Omron CX-Programmer project 新工程 (CX-Programmer 9.73)

# PLC 新PLC1: CPM2* 

## Global symbols (name address type ; comment)
0.00 BOOL  ; 横限1
0.01 BOOL  ; 横限2
0.02 BOOL  ; 横限3
0.03 BOOL  ; 横限4
0.04 BOOL  ; 横限5
0.05 BOOL  ; 二层上限1
0.06 BOOL  ; 二层上限2
0.07 BOOL  ; 二层上限3
0.08 BOOL  ; 二层上限4
0.09 BOOL  ; 二层下限1
0.10 BOOL  ; 二层下限2
0.11 BOOL  ; 二层下限3
10.00 BOOL  ; 总接触器1
10.01 BOOL  ; 总接触器2
10.02 BOOL  ; 1号可升降
10.03 BOOL  ; 2号可升降
10.04 BOOL  ; 3号可升降
10.06 BOOL  ; 4号可升降
11.00 BOOL  ; 5号横移
11.01 BOOL  ; 6号横移
11.02 BOOL  ; 7号横移
11.03 BOOL  ; 8号横移
11.04 BOOL  ; 9号可升降
11.06 BOOL  ; 10号可升降
12.00 BOOL  ; 11号可升降
12.01 BOOL  ; 12号可升降
12.02 BOOL  ; 故障报警
12.03 BOOL  ; 运行警示
12.04 BOOL  ; 左围栏升降
12.05 BOOL  ; 右围栏升降
12.06 BOOL  ; 围栏总上升
12.07 BOOL  ; 围栏总下降
16.00 BOOL  ; 手1
16.01 BOOL  ; 手2
16.02 BOOL  ; 手3
16.03 BOOL  ; 手4
16.04 BOOL  ; 手5
16.05 BOOL  ; 手6
16.06 BOOL  ; 手7
16.07 BOOL  ; 手8
16.08 BOOL  ; 手9
17.00 BOOL  ; 手动有车位输入
17.07 BOOL  ; =0
17.08 BOOL  ; >0
17.10 BOOL  ; OK
17.11 BOOL  ; ER
17.15 BOOL  ; >14
18.08 BOOL  ; 自动↑
18.09 BOOL  ; 手动↑
18.10 BOOL  ; 刷卡↑
18.13 BOOL  ; 启动延迟
18.14 BOOL  ; 自动脉冲
1.00 BOOL  ; 二层下限4
1.01 BOOL  ; 底层上限1
1.02 BOOL  ; 底层上限2
1.03 BOOL  ; 底层上限3
1.04 BOOL  ; 底层上限4
1.05 BOOL  ; 底层下限1
1.06 BOOL  ; 底层下限2
1.07 BOOL  ; 底层下限3
1.08 BOOL  ; 底层下限4
1.09 BOOL  ; 左围栏上限
1.10 BOOL  ; 右围栏上限
1.11 BOOL  ; 左围栏下限
202.01 BOOL  ; 1号卡
202.02 BOOL  ; 2号卡
202.03 BOOL  ; 3号卡
202.04 BOOL  ; 4号卡
202.05 BOOL  ; 5号卡
202.06 BOOL  ; 6号卡
202.07 BOOL  ; 7号卡
202.08 BOOL  ; 8号卡
202.09 BOOL  ; 9号卡
202.10 BOOL  ; 10号卡
202.11 BOOL  ; 11号卡
202.12 BOOL  ; 12号卡
203.02 BOOL  ; 二层可上
203.03 BOOL  ; 底层可下
203.05 BOOL  ; 二层全在上
203.06 BOOL  ; 底层全在下
203.07 BOOL  ; 升降至原位
204.00 BOOL  ; 0
204.01 BOOL  ; 1
204.02 BOOL  ; 2
204.03 BOOL  ; 3
204.04 BOOL  ; 4
204.05 BOOL  ; 5
204.06 BOOL  ; 6
204.07 BOOL  ; 7
204.08 BOOL  ; 8
204.09 BOOL  ; 9
205.04 BOOL  ; 升降
206.10 BOOL  ; 运行
206.11 BOOL  ; 故障
206.12 BOOL  ; 故障排除后启动
206.13 BOOL  ; 有故障
206.14 BOOL  ; 故障排除
206.15 BOOL  ; 故障↓
207.00 BOOL  ; 操作可
207.02 BOOL  ; 卡号
207.15 BOOL  ; 升降
208.00 BOOL  ; 自动车位号为1234
208.01 BOOL  ; 自动
208.02 BOOL  ; 在中间
208.05 BOOL  ; 自动车位号不等于1234
208.06 BOOL  ; 自动车位号不等于1234
208.07 BOOL  ; > 12
208.09 BOOL  ; ＞12，14
209.00 BOOL  ; 自动
209.01 BOOL  ; 手动
209.02 BOOL  ; 刷卡↑
209.05 BOOL  ; 刷卡
209.14 BOOL  ; 自动↑
209.15 BOOL  ; 自动车位号不等于1234↑
210.05 BOOL  ; 有四位数输入
211.00 BOOL  ; O-0
211.01 BOOL  ; 0-1
211.02 BOOL  ; 0-2
211.03 BOOL  ; 0-3
211.04 BOOL  ; 0-4
211.05 BOOL  ; 0-5
211.06 BOOL  ; 0-6
211.07 BOOL  ; 0-7
211.08 BOOL  ; 0-8
211.09 BOOL  ; 0-9
212.00 BOOL  ; 1-0
212.01 BOOL  ; 1-1
212.02 BOOL  ; 1-2
212.03 BOOL  ; 1-3
212.04 BOOL  ; 1-4
212.05 BOOL  ; 1-5
212.06 BOOL  ; 1-6
212.07 BOOL  ; 1-7
212.08 BOOL  ; 1-8
212.09 BOOL  ; 1-9
212.10 BOOL  ; F保持
212.11 BOOL  ; 左围栏S
212.12 BOOL  ; 右围栏S
213.00 BOOL  ; 2-0
213.01 BOOL  ; 2-1
213.02 BOOL  ; 2-2
213.03 BOOL  ; 2-3
213.04 BOOL  ; 2-4
213.05 BOOL  ; 2-5
213.06 BOOL  ; 2-6
213.07 BOOL  ; 2-7
213.08 BOOL  ; 2-8
213.09 BOOL  ; 2-9
213.11 BOOL  ; 左围栏X
213.12 BOOL  ; 右围栏X
214.00 BOOL  ; 3-0
214.01 BOOL  ; 3-1
214.02 BOOL  ; 3-2
214.03 BOOL  ; 3-3
214.04 BOOL  ; 3-4
214.05 BOOL  ; 3-5
214.06 BOOL  ; 3-6
214.07 BOOL  ; 3-7
214.08 BOOL  ; 3-8
214.09 BOOL  ; 3-9
216.01 BOOL  ; 1号卡2
216.02 BOOL  ; 2号卡2
216.03 BOOL  ; 3号卡2
216.04 BOOL  ; 4号卡2
216.05 BOOL  ; 5号卡2
216.06 BOOL  ; 6号卡2
216.07 BOOL  ; 7号卡2
216.08 BOOL  ; 8号卡2
216.09 BOOL  ; 9号卡2
216.10 BOOL  ; 10号卡2
216.11 BOOL  ; 11号卡2
216.12 BOOL  ; 12号卡2
217.00 BOOL  ; 升降至原位↑
217.01 BOOL  ; 到位
219.01 BOOL  ; 1号卡3
219.02 BOOL  ; 2号卡3
219.03 BOOL  ; 3号卡3
219.04 BOOL  ; 4号卡3
219.05 BOOL  ; 5号卡3
219.06 BOOL  ; 6号卡3
219.07 BOOL  ; 7号卡3
219.08 BOOL  ; 8号卡3
219.09 BOOL  ; 9号卡3
219.10 BOOL  ; 10号卡3
219.11 BOOL  ; 11号卡3
219.12 BOOL  ; 12号卡3
220.10 BOOL  ; 一位输入
220.11 BOOL  ; 二位输入
220.12 BOOL  ; 三位输入
220.13 BOOL  ; 四位输入
222.00 BOOL  ; 手10
222.01 BOOL  ; 手11
222.02 BOOL  ; 手12
222.03 BOOL  ; 手13
222.04 BOOL  ; 手14
224.00 BOOL  ; 手取1
224.01 BOOL  ; 手取2
224.02 BOOL  ; 手取3
224.03 BOOL  ; 手取4
224.04 BOOL  ; 手取5
224.05 BOOL  ; 手取6
224.06 BOOL  ; 手取7
224.07 BOOL  ; 手取8
224.08 BOOL  ; 手取9
224.09 BOOL  ; 手取10
224.10 BOOL  ; 手取11
224.12 BOOL  ; 手取12
224.13 BOOL  ; 手取13
224.14 BOOL  ; 手取14
22.00 BOOL  ; 横移过快
22.01 BOOL  ; 有故障
22.02 BOOL  ; 横移过快
22.06 BOOL  ; 横移
22.07 BOOL  ; 5号横移↓
22.08 BOOL  ; 6号横移↓
22.09 BOOL  ; 7号横移↓
22.10 BOOL  ; 8号横移↓
22.11 BOOL  ; 人车进出上升沿
22.12 BOOL  ; 延时上升沿
230.06 BOOL  ; 7Z
230.07 BOOL  ; 5Z
230.08 BOOL  ; 6Z
230.09 BOOL  ; 7Z
230.10 BOOL  ; 8Z
230.12 BOOL  ; 12Z
232.00 BOOL  ; 1S
232.01 BOOL  ; 2S
232.02 BOOL  ; 3S
232.03 BOOL  ; 4S
232.14 BOOL  ; 9S
232.15 BOOL  ; 10S
233.00 BOOL  ; 11S
233.01 BOOL  ; 12S
236.00 BOOL  ; ZD1
236.01 BOOL  ; ZD2
236.02 BOOL  ; ZD3
236.03 BOOL  ; ZD4
236.05 BOOL  ; ZD6
236.06 BOOL  ; ZD7
236.07 BOOL  ; ZD9
236.08 BOOL  ; ZD10
236.09 BOOL  ; ZD11
236.10 BOOL  ; ZD12
23.00 BOOL  ; 横移
23.01 BOOL  ; 横移
240.07 BOOL  ; 5Y
240.08 BOOL  ; 6Y
240.09 BOOL  ; 7Y
240.10 BOOL  ; 8Y
242.00 BOOL  ; 1X
242.01 BOOL  ; 2X
242.02 BOOL  ; 3X
242.03 BOOL  ; 4X
242.14 BOOL  ; 9X
242.15 BOOL  ; 10X
243.00 BOOL  ; 11X
243.01 BOOL  ; 12X
28.08 BOOL  ; > 14
2.00 BOOL  ; 右围栏下限
2.01 BOOL  ; 底层防坠落
2.02 BOOL  ; 二层松链
2.03 BOOL  ; 底层超上限
2.04 BOOL  ; 二层超上限
2.05 BOOL  ; 车高光电
2.06 BOOL  ; 人车进出
2.07 BOOL  ; 车长光电
2.08 BOOL  ; 急停
2.09 BOOL  ; 热保护
2.10 BOOL  ; 相序保护
30.00 BOOL  ; 1号在下
30.01 BOOL  ; 2号在下
30.02 BOOL  ; 3号在下
30.03 BOOL  ; 4号在下
31.01 BOOL  ; 二层总上升
31.02 BOOL  ; 二层总下降
31.03 BOOL  ; 底层总上升
31.04 BOOL  ; 底层总下降
31.05 BOOL  ; 一层总左移
31.06 BOOL  ; 一层总右移
31.07 BOOL  ; 左围栏上升
31.08 BOOL  ; 左围栏下降
31.09 BOOL  ; 右围栏上升
31.10 BOOL  ; 右围栏下降
32.02 BOOL  ; （到位）
34.00 BOOL  ; Z1
34.01 BOOL  ; Z2
34.02 BOOL  ; Z3
34.03 BOOL  ; Z4
34.04 BOOL  ; Z5
34.05 BOOL  ; Z6
34.06 BOOL  ; Z7
34.07 BOOL  ; Z8
34.08 BOOL  ; Z9
34.09 BOOL  ; Z10
34.10 BOOL  ; Z11
34.12 BOOL  ; Z12
35.15 BOOL  ; > 12
37.12 BOOL  ; 重取
40.00 BOOL  ; 0
40.01 BOOL  ; 1
40.02 BOOL  ; 2/上
40.03 BOOL  ; 3
40.04 BOOL  ; 4左
40.05 BOOL  ; 5
40.06 BOOL  ; 6右
40.07 BOOL  ; 7
40.08 BOOL  ; 8/下
40.09 BOOL  ; 9
40.10 BOOL  ; 启动
40.11 BOOL  ; 复位
40.12 BOOL  ; 手动
40.13 BOOL  ; 在中间
40.14 BOOL  ; 自动
40.15 BOOL  ; F
41.00 BOOL  ; 1号可上下
41.01 BOOL  ; 2号可上下
41.02 BOOL  ; 3号可上下
41.03 BOOL  ; 4号可上下
41.08 BOOL  ; 9号可上下
41.09 BOOL  ; 10号可上下
41.10 BOOL  ; 11号可上下
41.11 BOOL  ; 12号可上下
42.01 BOOL  ; 1号卡
42.02 BOOL  ; 2号卡
42.03 BOOL  ; 3号卡
42.04 BOOL  ; 4号卡
42.05 BOOL  ; 5号卡
42.06 BOOL  ; 6号卡
42.07 BOOL  ; 7号卡
42.08 BOOL  ; 8号卡
43.00 BOOL  ; 9号卡
43.01 BOOL  ; 10号卡
43.02 BOOL  ; 11号卡
43.03 BOOL  ; 12号卡
44.01 BOOL  ; 1号卡2
44.02 BOOL  ; 2号卡2
44.03 BOOL  ; 3号卡2
44.04 BOOL  ; 4号卡2
44.05 BOOL  ; 5号卡2
44.06 BOOL  ; 6号卡2
44.07 BOOL  ; 7号卡2
44.08 BOOL  ; 8号卡2
45.00 BOOL  ; 9号卡2
45.01 BOOL  ; 10号卡2
45.02 BOOL  ; 11号卡2
45.03 BOOL  ; 12号卡2
46.01 BOOL  ; 1号卡3
46.02 BOOL  ; 2号卡3
46.03 BOOL  ; 3号卡3
46.04 BOOL  ; 4号卡3
46.05 BOOL  ; 5号卡3
46.06 BOOL  ; 6号卡3
46.07 BOOL  ; 7号卡3
46.08 BOOL  ; 8号卡3
47.00 BOOL  ; 9号卡3
47.01 BOOL  ; 10号卡3
47.02 BOOL  ; 11号卡3
47.03 BOOL  ; 12号卡3
48.00 BOOL  ; 左围上
48.01 BOOL  ; 右围上
48.02 BOOL  ; 左围下
48.03 BOOL  ; 右围下
CNT011 BOOL  ; 二层升降计时
CNT012 BOOL  ; 底层升降计时
CNT013 BOOL  ; 计数
CNT014 BOOL  ; 计数
CNT077 BOOL  ; 横移计时
CNT078 BOOL  ; 围栏上升计时
CNT079 BOOL  ; 围栏下降计时
DM10 CHANNEL  ; 刷卡密码1
DM100 CHANNEL  ; 故障代码
DM11 CHANNEL  ; 刷卡密码2
DM12 CHANNEL  ; 刷卡密码3
DM13 CHANNEL  ; 刷卡密码4
DM14 CHANNEL  ; 刷卡密码5
DM20 CHANNEL  ; 1位
DM21 CHANNEL  ; 2位
DM22 CHANNEL  ; 3位
DM23 CHANNEL  ; 4位
DM8 CHANNEL  ; 自动车位
DM9 CHANNEL  ; 手动号码
HR0.00 BOOL  ; 保持
HR0.01 BOOL  ; 保持
HR0.02 BOOL  ; 保持
TIM020 BOOL  ; 启动延时
TIM036 BOOL  ; 延时
TIM044 BOOL  ; 0.8
TIM045 BOOL  ; 延时
TIM046 BOOL  ; 延时
TIM047 BOOL  ; 延迟
TIM050 BOOL  ; 延迟
TIM051 BOOL  ; 延迟

## Program 新程序1 (no task)
; 这是我为“杭州三层下一A12停车场”设计的立体车库系统，底层设有12个车位，配备三层结构、刷卡功能和围栏控制，用户可通过刷卡或手动操作存取车辆。 / 系统设备包括PLC控制器、刷卡器、数字键、围栏升降装置、升降机构、横移机构、故障检测传感器和报警装置。 / 系统启动时，用户刷卡后输入刷卡密码1-5的五位密码，验证通过后置位对应卡验证标志，如1号卡验证标志表示第1号卡可用，允许进入操作流程。 / 在自动模式下，用户通过数字键0-9输入车位号，存储至车位号第1-4位，并由自动车位号记录目标车位。 / 在手动模式下，用户通过手动模式开关输入手动车位号。 / 在自动或手动模式下，自动车位号和手动车位号的值需为1到12，若超出范围，故障代码存储记录错误，系统暂停升降和横移动作。 / 按下启动按钮后，系统根据二层可上升标志和底层可下降标志判断目标车位状态。 / 若车位空闲，系统启动相应动作，如通过二层总上升控制提升二层，或通过一层总左移控制调整一层位置。 / 为避免机械冲突，二层总上升控制、二层总下降控制、底层总上升控制、底层总下降控制与一层总左移控制、一层总右移控制不可同时激活。 / 为防止升降机构冲突，二层总上升控制与二层总下降控制不可同时动作，底层总上升控制与底层总下降控制亦不可同时动作。 / 为避免横移机构冲突，一层总左移控制与一层总右移控制不可同时动作。 / 车辆进出时，围栏总上升控制和围栏总下降控制调整围栏位置，需左围栏上限传感器或右围栏上限传感器确认到位后，方可启动二层总上升控制、二层总下降控制、底层总上升控制、底层总下降控制、一层总左移控制或一层总右移控制。 / 当车位号有效且围栏需下降时，激活围栏总下降控制。当左围栏上限传感器检测到位时，允许围栏总上升控制动作。当右围栏上限传感器检测到位时，允许围栏总下降控制动作。 / 系统实时监控故障信号，如急停按钮触发时，故障代码存储置为55，故障报警灯亮起，所有升降和横移动作停止。 / 若故障代码存储不为0，表明存在未排除故障，二层总上升控制、二层总下降控制、底层总上升控制、底层总下降控制、一层总左移控制、一层总右移控制不可启动，直至按下复位按钮清零故障代码。 / 运行中，运行警示灯点亮提示操作状态，系统通过定时器（如TIM020）设置启动延时，确保动作顺序正确。

### Section 段1

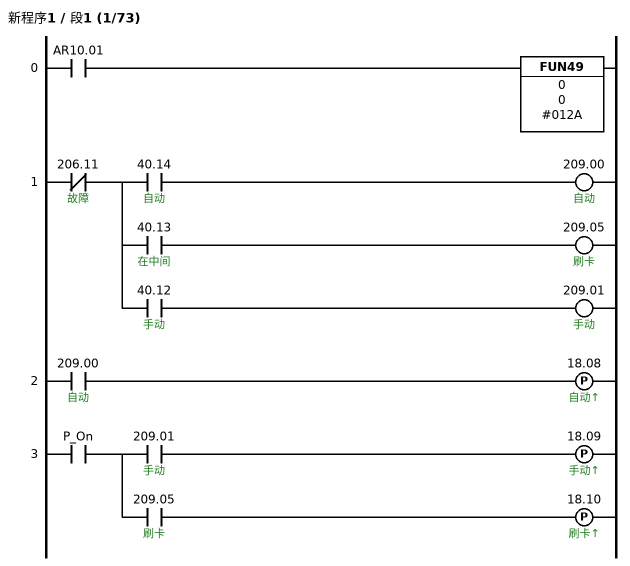
; rung 0
LD AR10.01
FUN49 0 0 #012A
; rung 1
LDNOT 206.11  ; 故障
OUT TR0
AND 40.14  ; 自动
OUT 209.00  ; 自动
LD TR0
AND 40.13  ; 在中间
OUT 209.05  ; 刷卡
LD TR0
AND 40.12  ; 手动
OUT 209.01  ; 手动
; rung 2
LD 209.00  ; 自动
DIFU(13) 18.08  ; 自动↑
; rung 3
LD P_On
OUT TR0
AND 209.01  ; 手动
DIFU(13) 18.09  ; 手动↑
LD TR0
AND 209.05  ; 刷卡
DIFU(13) 18.10  ; 刷卡↑

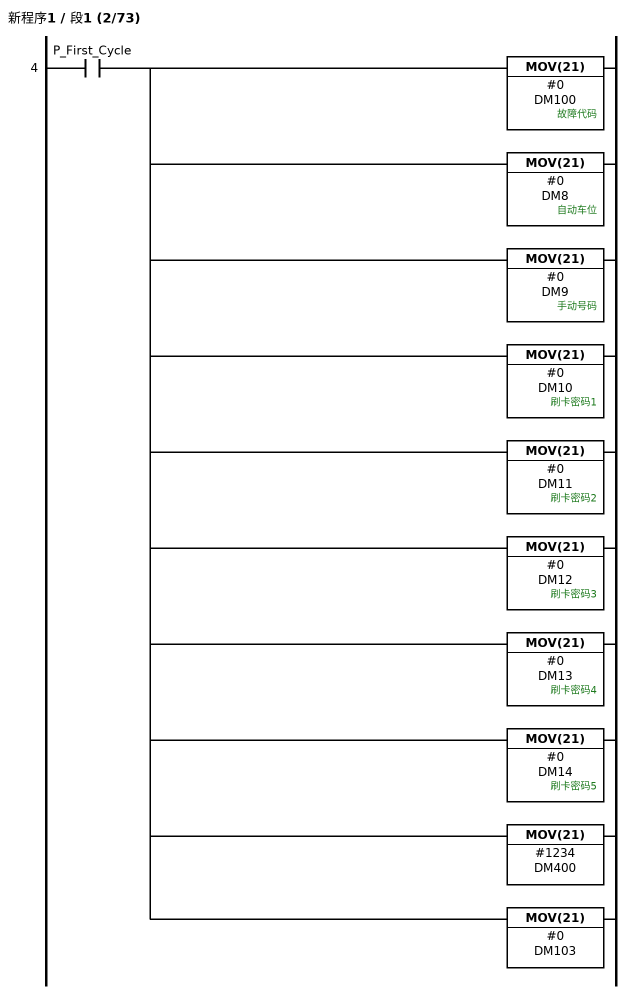
; rung 4
LD P_First_Cycle
MOV(21) #0 DM100  ; 故障代码
MOV(21) #0 DM8  ; 自动车位
MOV(21) #0 DM9  ; 手动号码
MOV(21) #0 DM10  ; 刷卡密码1
MOV(21) #0 DM11  ; 刷卡密码2
MOV(21) #0 DM12  ; 刷卡密码3
MOV(21) #0 DM13  ; 刷卡密码4
MOV(21) #0 DM14  ; 刷卡密码5
MOV(21) #1234 DM400
MOV(21) #0 DM103

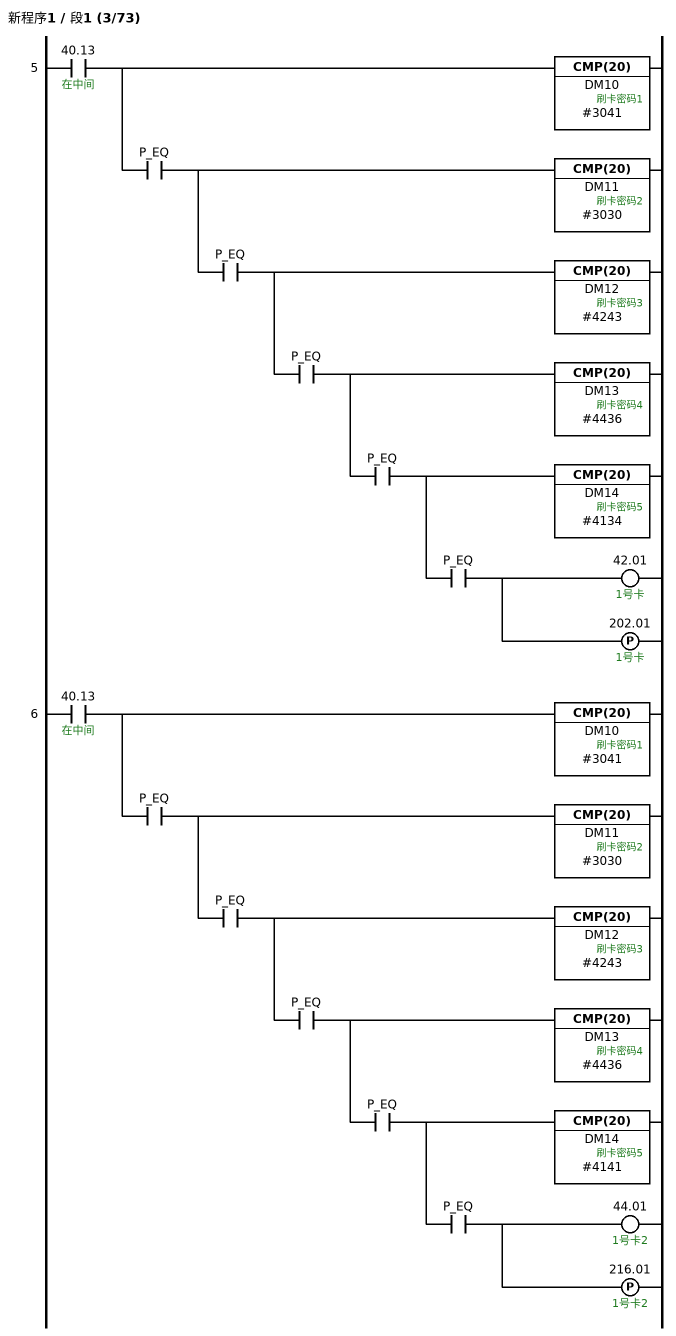
; rung 5
LD 40.13  ; 在中间
CMP(20) DM10 #3041  ; 刷卡密码1
AND P_EQ
CMP(20) DM11 #3030  ; 刷卡密码2
AND P_EQ
CMP(20) DM12 #4243  ; 刷卡密码3
AND P_EQ
CMP(20) DM13 #4436  ; 刷卡密码4
AND P_EQ
CMP(20) DM14 #4134  ; 刷卡密码5
AND P_EQ
OUT 42.01  ; 1号卡
DIFU(13) 202.01  ; 1号卡
; rung 6
LD 40.13  ; 在中间
CMP(20) DM10 #3041  ; 刷卡密码1
AND P_EQ
CMP(20) DM11 #3030  ; 刷卡密码2
AND P_EQ
CMP(20) DM12 #4243  ; 刷卡密码3
AND P_EQ
CMP(20) DM13 #4436  ; 刷卡密码4
AND P_EQ
CMP(20) DM14 #4141  ; 刷卡密码5
AND P_EQ
OUT 44.01  ; 1号卡2
DIFU(13) 216.01  ; 1号卡2

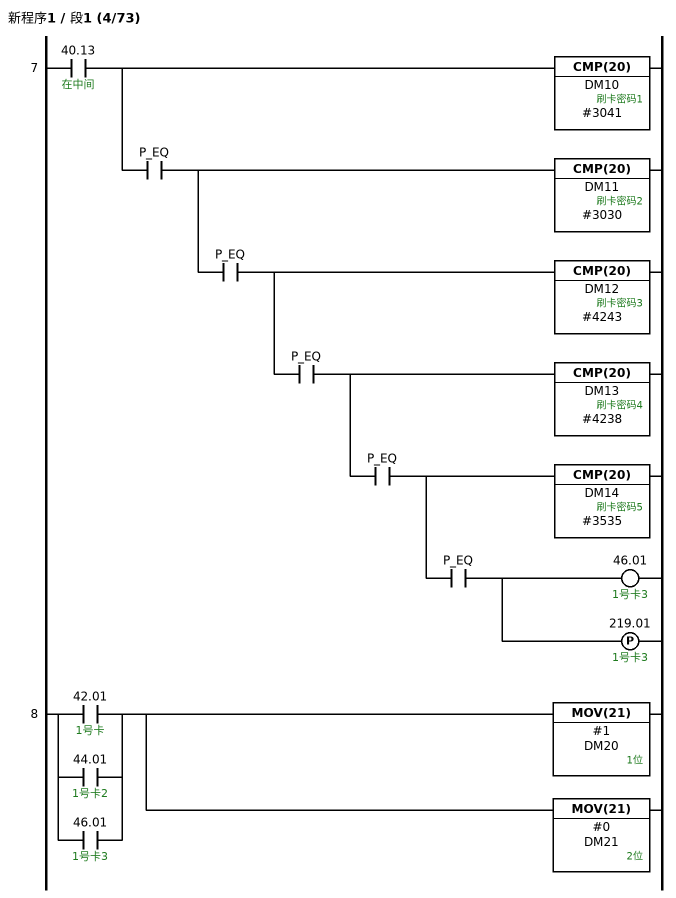
; rung 7
LD 40.13  ; 在中间
CMP(20) DM10 #3041  ; 刷卡密码1
AND P_EQ
CMP(20) DM11 #3030  ; 刷卡密码2
AND P_EQ
CMP(20) DM12 #4243  ; 刷卡密码3
AND P_EQ
CMP(20) DM13 #4238  ; 刷卡密码4
AND P_EQ
CMP(20) DM14 #3535  ; 刷卡密码5
AND P_EQ
OUT 46.01  ; 1号卡3
DIFU(13) 219.01  ; 1号卡3
; rung 8
LD 42.01  ; 1号卡
OR 44.01  ; 1号卡2
OR 46.01  ; 1号卡3
MOV(21) #1 DM20  ; 1位
MOV(21) #0 DM21  ; 2位

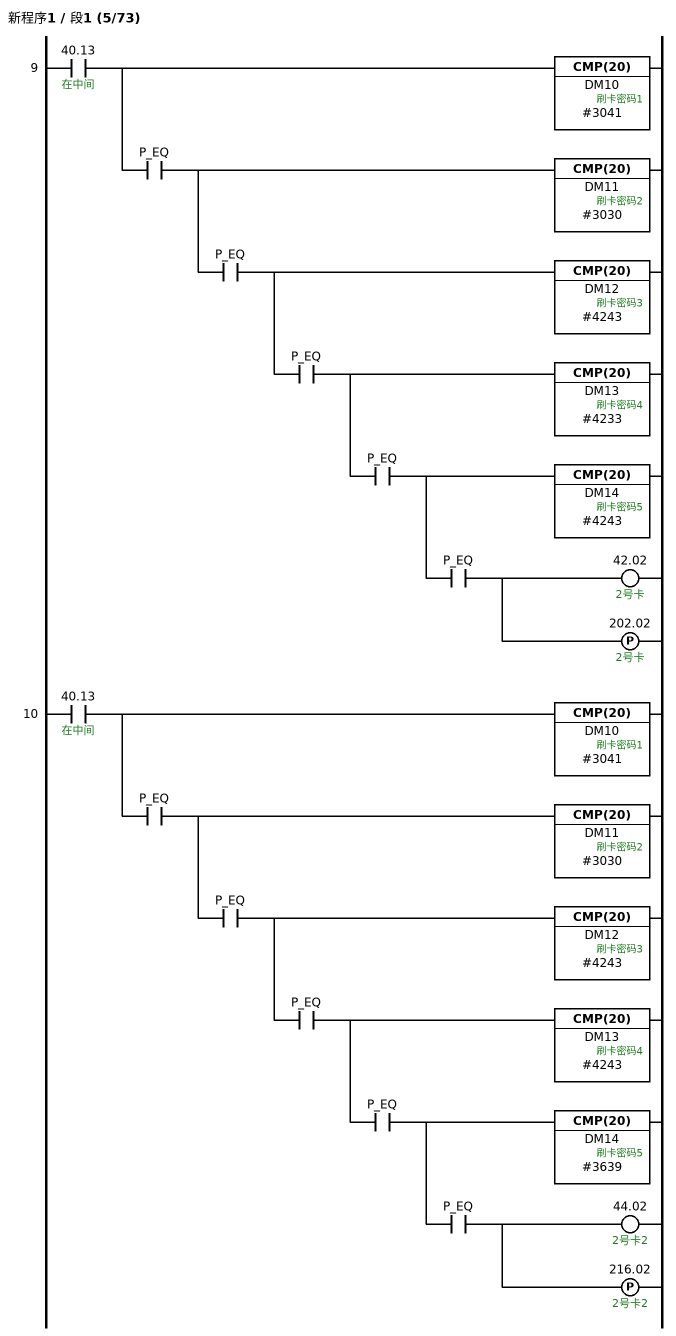
; rung 9
LD 40.13  ; 在中间
CMP(20) DM10 #3041  ; 刷卡密码1
AND P_EQ
CMP(20) DM11 #3030  ; 刷卡密码2
AND P_EQ
CMP(20) DM12 #4243  ; 刷卡密码3
AND P_EQ
CMP(20) DM13 #4233  ; 刷卡密码4
AND P_EQ
CMP(20) DM14 #4243  ; 刷卡密码5
AND P_EQ
OUT 42.02  ; 2号卡
DIFU(13) 202.02  ; 2号卡
; rung 10
LD 40.13  ; 在中间
CMP(20) DM10 #3041  ; 刷卡密码1
AND P_EQ
CMP(20) DM11 #3030  ; 刷卡密码2
AND P_EQ
CMP(20) DM12 #4243  ; 刷卡密码3
AND P_EQ
CMP(20) DM13 #4243  ; 刷卡密码4
AND P_EQ
CMP(20) DM14 #3639  ; 刷卡密码5
AND P_EQ
OUT 44.02  ; 2号卡2
DIFU(13) 216.02  ; 2号卡2

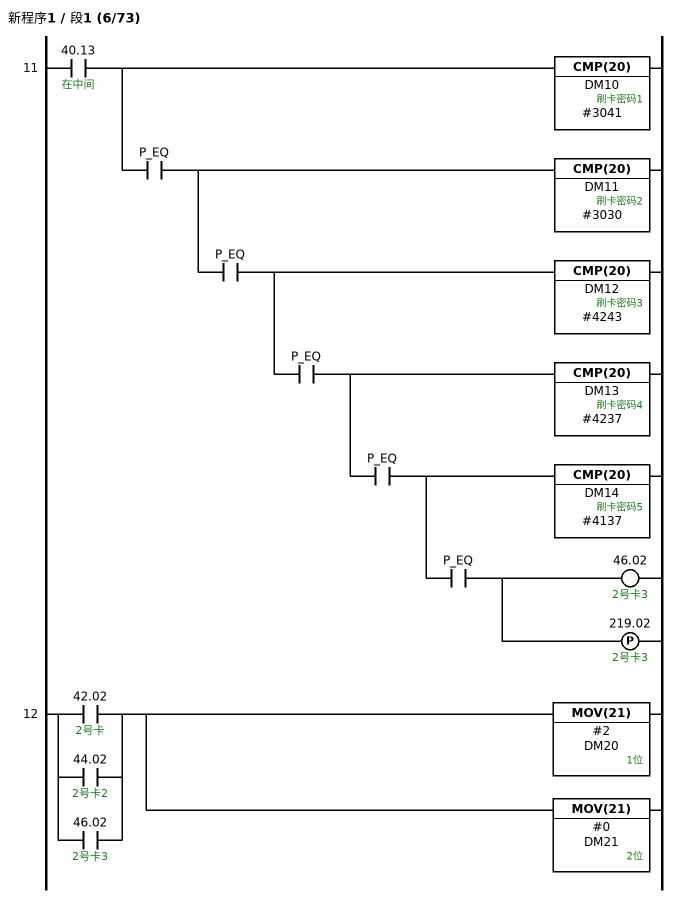
; rung 11
LD 40.13  ; 在中间
CMP(20) DM10 #3041  ; 刷卡密码1
AND P_EQ
CMP(20) DM11 #3030  ; 刷卡密码2
AND P_EQ
CMP(20) DM12 #4243  ; 刷卡密码3
AND P_EQ
CMP(20) DM13 #4237  ; 刷卡密码4
AND P_EQ
CMP(20) DM14 #4137  ; 刷卡密码5
AND P_EQ
OUT 46.02  ; 2号卡3
DIFU(13) 219.02  ; 2号卡3
; rung 12
LD 42.02  ; 2号卡
OR 44.02  ; 2号卡2
OR 46.02  ; 2号卡3
MOV(21) #2 DM20  ; 1位
MOV(21) #0 DM21  ; 2位

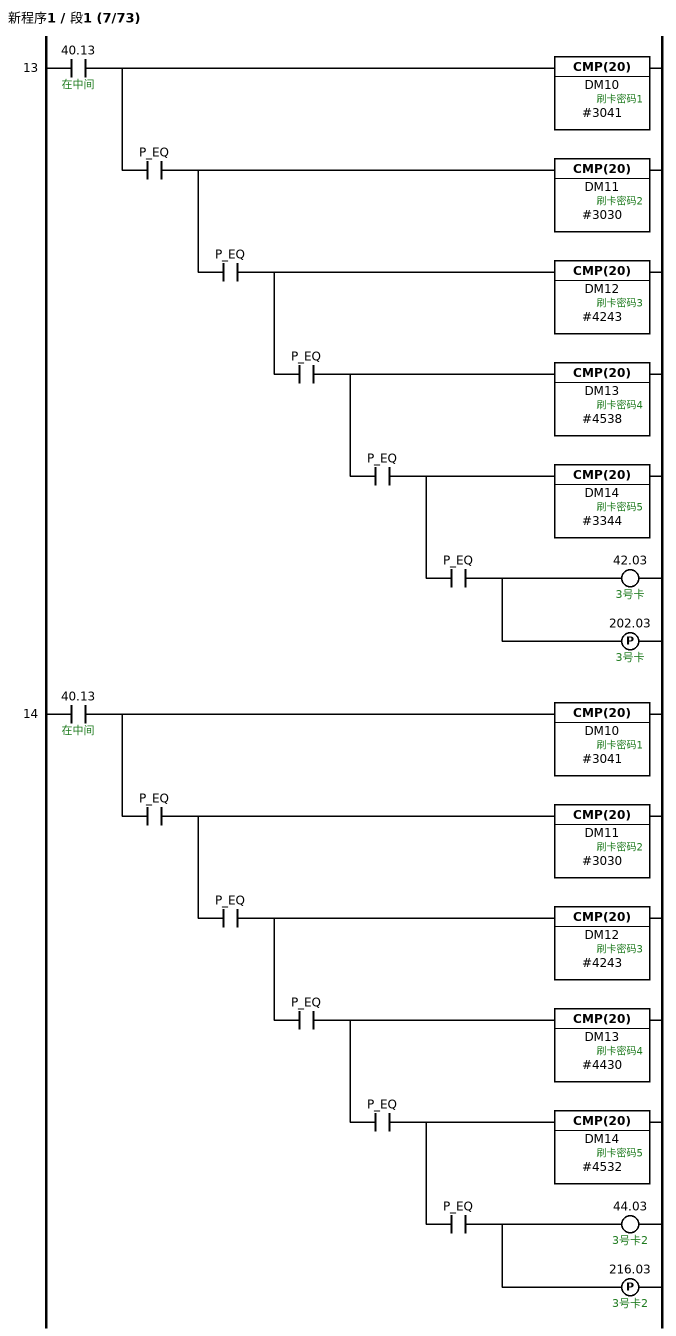
; rung 13
LD 40.13  ; 在中间
CMP(20) DM10 #3041  ; 刷卡密码1
AND P_EQ
CMP(20) DM11 #3030  ; 刷卡密码2
AND P_EQ
CMP(20) DM12 #4243  ; 刷卡密码3
AND P_EQ
CMP(20) DM13 #4538  ; 刷卡密码4
AND P_EQ
CMP(20) DM14 #3344  ; 刷卡密码5
AND P_EQ
OUT 42.03  ; 3号卡
DIFU(13) 202.03  ; 3号卡
; rung 14
LD 40.13  ; 在中间
CMP(20) DM10 #3041  ; 刷卡密码1
AND P_EQ
CMP(20) DM11 #3030  ; 刷卡密码2
AND P_EQ
CMP(20) DM12 #4243  ; 刷卡密码3
AND P_EQ
CMP(20) DM13 #4430  ; 刷卡密码4
AND P_EQ
CMP(20) DM14 #4532  ; 刷卡密码5
AND P_EQ
OUT 44.03  ; 3号卡2
DIFU(13) 216.03  ; 3号卡2

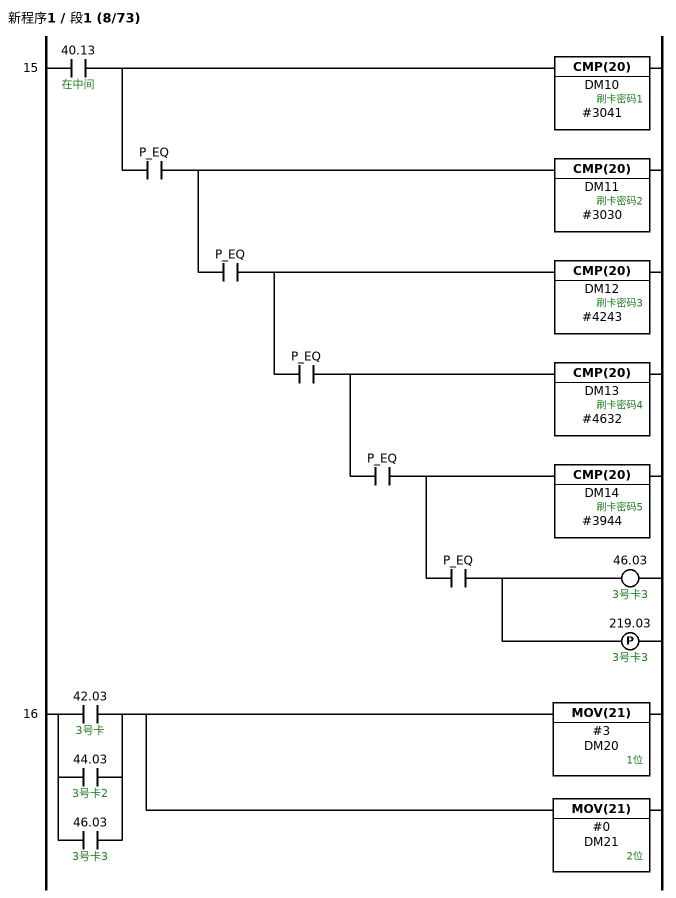
; rung 15
LD 40.13  ; 在中间
CMP(20) DM10 #3041  ; 刷卡密码1
AND P_EQ
CMP(20) DM11 #3030  ; 刷卡密码2
AND P_EQ
CMP(20) DM12 #4243  ; 刷卡密码3
AND P_EQ
CMP(20) DM13 #4632  ; 刷卡密码4
AND P_EQ
CMP(20) DM14 #3944  ; 刷卡密码5
AND P_EQ
OUT 46.03  ; 3号卡3
DIFU(13) 219.03  ; 3号卡3
; rung 16
LD 42.03  ; 3号卡
OR 44.03  ; 3号卡2
OR 46.03  ; 3号卡3
MOV(21) #3 DM20  ; 1位
MOV(21) #0 DM21  ; 2位

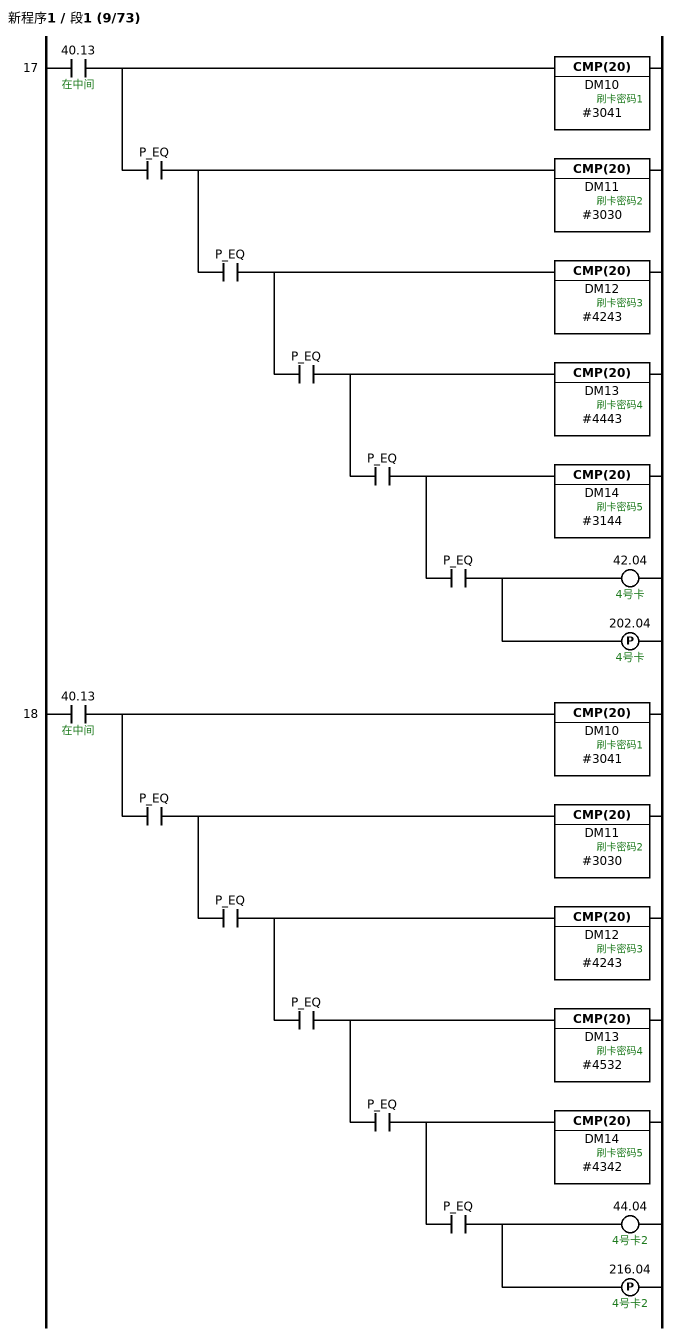
; rung 17
LD 40.13  ; 在中间
CMP(20) DM10 #3041  ; 刷卡密码1
AND P_EQ
CMP(20) DM11 #3030  ; 刷卡密码2
AND P_EQ
CMP(20) DM12 #4243  ; 刷卡密码3
AND P_EQ
CMP(20) DM13 #4443  ; 刷卡密码4
AND P_EQ
CMP(20) DM14 #3144  ; 刷卡密码5
AND P_EQ
OUT 42.04  ; 4号卡
DIFU(13) 202.04  ; 4号卡
; rung 18
LD 40.13  ; 在中间
CMP(20) DM10 #3041  ; 刷卡密码1
AND P_EQ
CMP(20) DM11 #3030  ; 刷卡密码2
AND P_EQ
CMP(20) DM12 #4243  ; 刷卡密码3
AND P_EQ
CMP(20) DM13 #4532  ; 刷卡密码4
AND P_EQ
CMP(20) DM14 #4342  ; 刷卡密码5
AND P_EQ
OUT 44.04  ; 4号卡2
DIFU(13) 216.04  ; 4号卡2

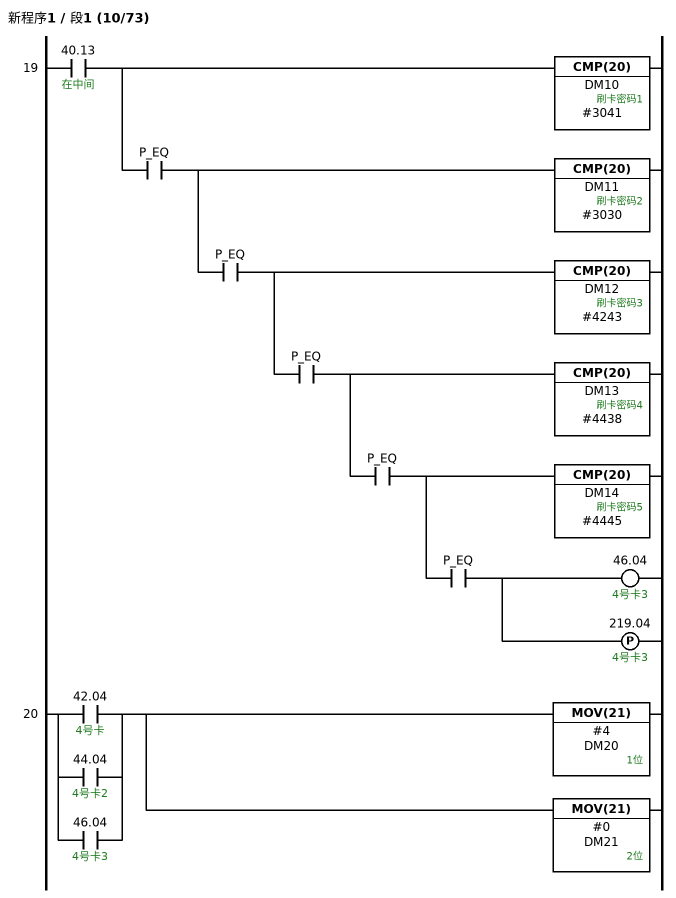
; rung 19
LD 40.13  ; 在中间
CMP(20) DM10 #3041  ; 刷卡密码1
AND P_EQ
CMP(20) DM11 #3030  ; 刷卡密码2
AND P_EQ
CMP(20) DM12 #4243  ; 刷卡密码3
AND P_EQ
CMP(20) DM13 #4438  ; 刷卡密码4
AND P_EQ
CMP(20) DM14 #4445  ; 刷卡密码5
AND P_EQ
OUT 46.04  ; 4号卡3
DIFU(13) 219.04  ; 4号卡3
; rung 20
LD 42.04  ; 4号卡
OR 44.04  ; 4号卡2
OR 46.04  ; 4号卡3
MOV(21) #4 DM20  ; 1位
MOV(21) #0 DM21  ; 2位

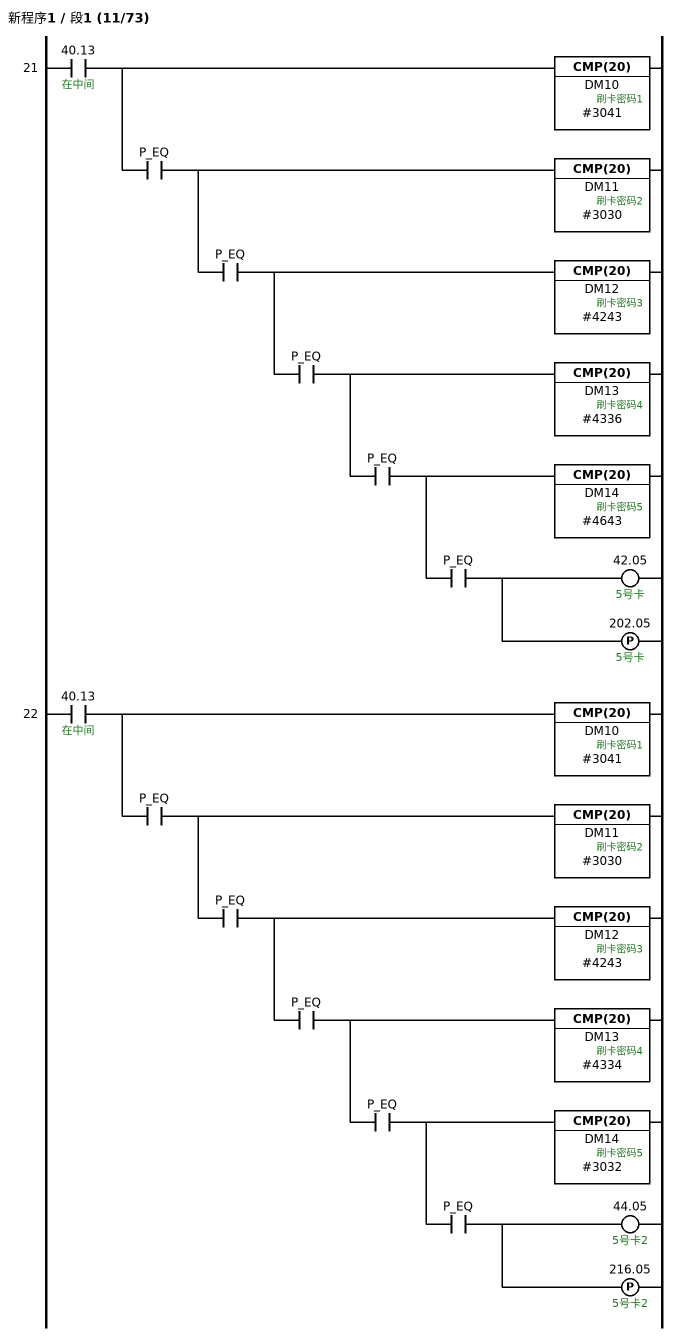
; rung 21
LD 40.13  ; 在中间
CMP(20) DM10 #3041  ; 刷卡密码1
AND P_EQ
CMP(20) DM11 #3030  ; 刷卡密码2
AND P_EQ
CMP(20) DM12 #4243  ; 刷卡密码3
AND P_EQ
CMP(20) DM13 #4336  ; 刷卡密码4
AND P_EQ
CMP(20) DM14 #4643  ; 刷卡密码5
AND P_EQ
OUT 42.05  ; 5号卡
DIFU(13) 202.05  ; 5号卡
; rung 22
LD 40.13  ; 在中间
CMP(20) DM10 #3041  ; 刷卡密码1
AND P_EQ
CMP(20) DM11 #3030  ; 刷卡密码2
AND P_EQ
CMP(20) DM12 #4243  ; 刷卡密码3
AND P_EQ
CMP(20) DM13 #4334  ; 刷卡密码4
AND P_EQ
CMP(20) DM14 #3032  ; 刷卡密码5
AND P_EQ
OUT 44.05  ; 5号卡2
DIFU(13) 216.05  ; 5号卡2

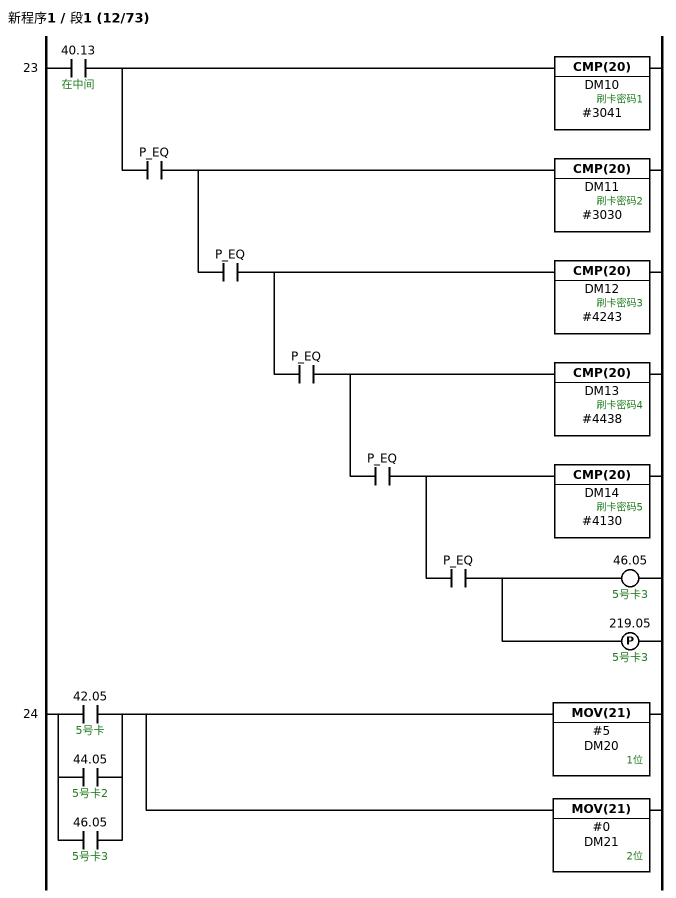
; rung 23
LD 40.13  ; 在中间
CMP(20) DM10 #3041  ; 刷卡密码1
AND P_EQ
CMP(20) DM11 #3030  ; 刷卡密码2
AND P_EQ
CMP(20) DM12 #4243  ; 刷卡密码3
AND P_EQ
CMP(20) DM13 #4438  ; 刷卡密码4
AND P_EQ
CMP(20) DM14 #4130  ; 刷卡密码5
AND P_EQ
OUT 46.05  ; 5号卡3
DIFU(13) 219.05  ; 5号卡3
; rung 24
LD 42.05  ; 5号卡
OR 44.05  ; 5号卡2
OR 46.05  ; 5号卡3
MOV(21) #5 DM20  ; 1位
MOV(21) #0 DM21  ; 2位

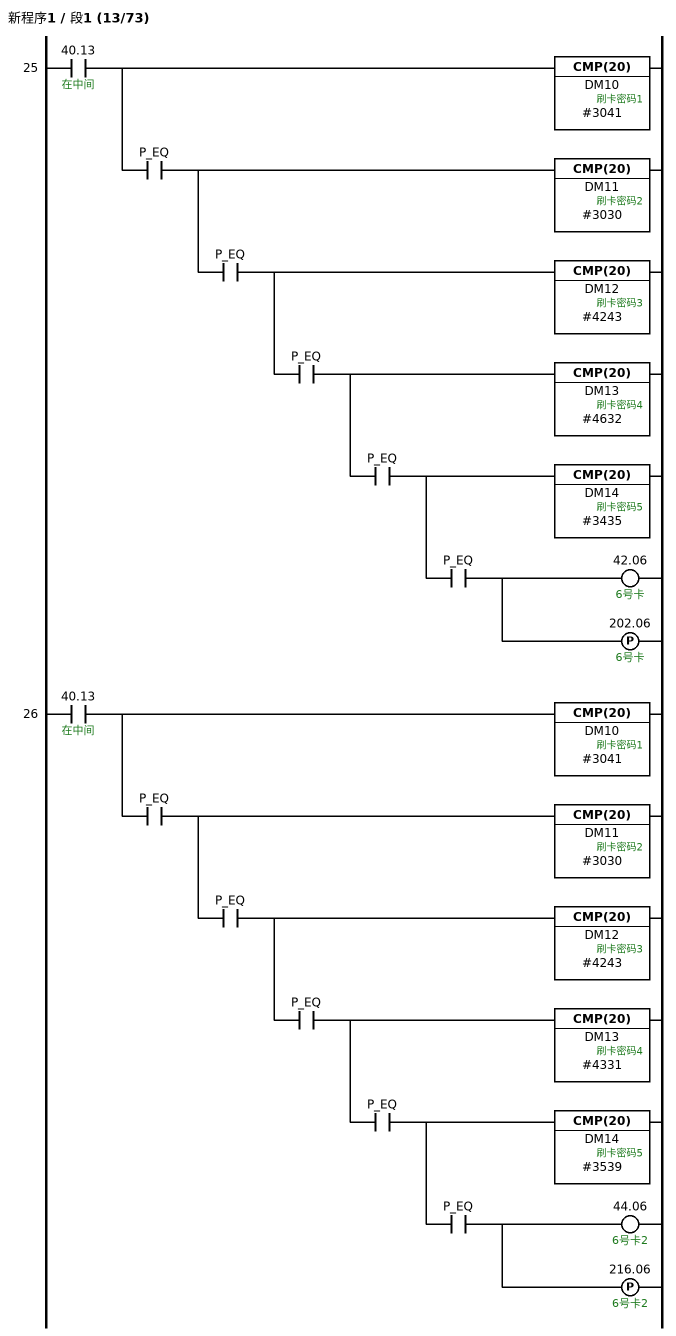
; rung 25
LD 40.13  ; 在中间
CMP(20) DM10 #3041  ; 刷卡密码1
AND P_EQ
CMP(20) DM11 #3030  ; 刷卡密码2
AND P_EQ
CMP(20) DM12 #4243  ; 刷卡密码3
AND P_EQ
CMP(20) DM13 #4632  ; 刷卡密码4
AND P_EQ
CMP(20) DM14 #3435  ; 刷卡密码5
AND P_EQ
OUT 42.06  ; 6号卡
DIFU(13) 202.06  ; 6号卡
; rung 26
LD 40.13  ; 在中间
CMP(20) DM10 #3041  ; 刷卡密码1
AND P_EQ
CMP(20) DM11 #3030  ; 刷卡密码2
AND P_EQ
CMP(20) DM12 #4243  ; 刷卡密码3
AND P_EQ
CMP(20) DM13 #4331  ; 刷卡密码4
AND P_EQ
CMP(20) DM14 #3539  ; 刷卡密码5
AND P_EQ
OUT 44.06  ; 6号卡2
DIFU(13) 216.06  ; 6号卡2

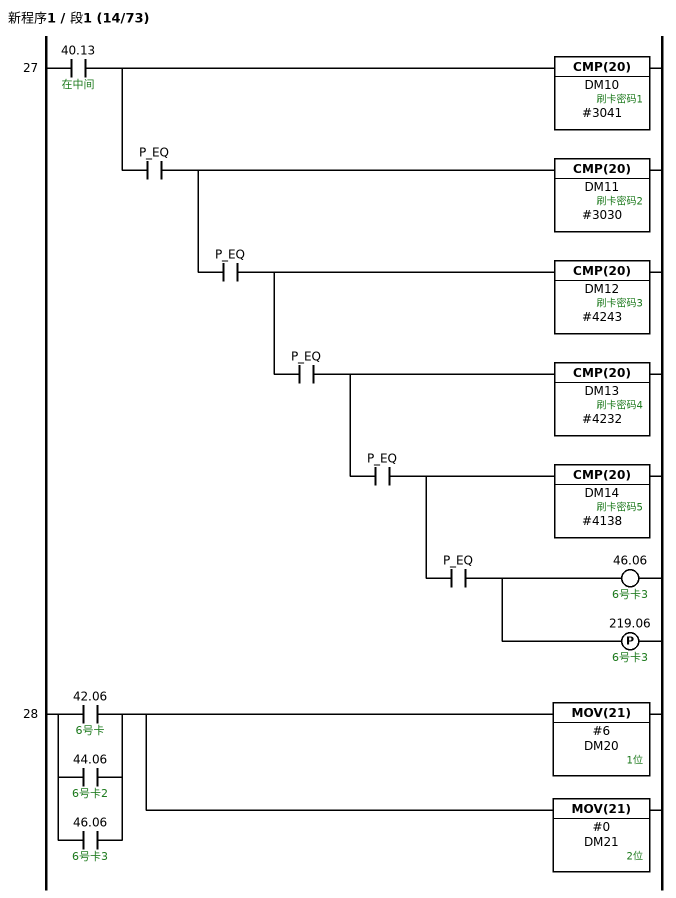
; rung 27
LD 40.13  ; 在中间
CMP(20) DM10 #3041  ; 刷卡密码1
AND P_EQ
CMP(20) DM11 #3030  ; 刷卡密码2
AND P_EQ
CMP(20) DM12 #4243  ; 刷卡密码3
AND P_EQ
CMP(20) DM13 #4232  ; 刷卡密码4
AND P_EQ
CMP(20) DM14 #4138  ; 刷卡密码5
AND P_EQ
OUT 46.06  ; 6号卡3
DIFU(13) 219.06  ; 6号卡3
; rung 28
LD 42.06  ; 6号卡
OR 44.06  ; 6号卡2
OR 46.06  ; 6号卡3
MOV(21) #6 DM20  ; 1位
MOV(21) #0 DM21  ; 2位

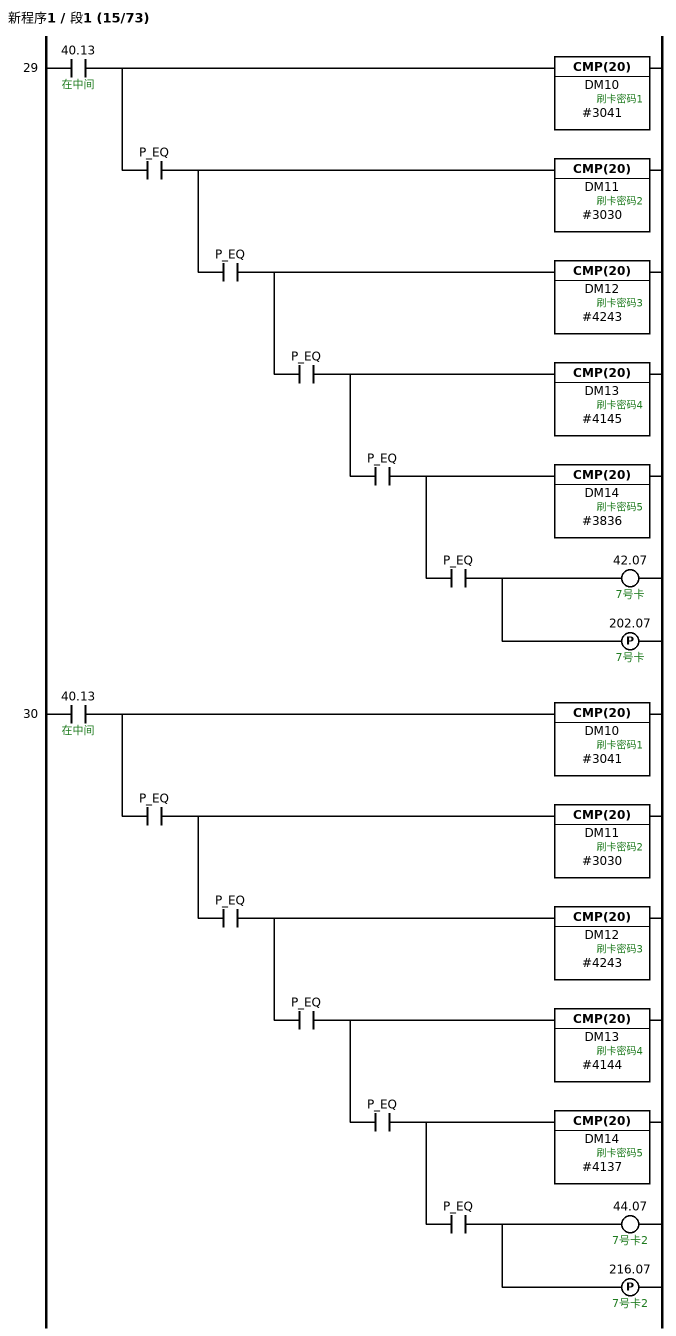
; rung 29
LD 40.13  ; 在中间
CMP(20) DM10 #3041  ; 刷卡密码1
AND P_EQ
CMP(20) DM11 #3030  ; 刷卡密码2
AND P_EQ
CMP(20) DM12 #4243  ; 刷卡密码3
AND P_EQ
CMP(20) DM13 #4145  ; 刷卡密码4
AND P_EQ
CMP(20) DM14 #3836  ; 刷卡密码5
AND P_EQ
OUT 42.07  ; 7号卡
DIFU(13) 202.07  ; 7号卡
; rung 30
LD 40.13  ; 在中间
CMP(20) DM10 #3041  ; 刷卡密码1
AND P_EQ
CMP(20) DM11 #3030  ; 刷卡密码2
AND P_EQ
CMP(20) DM12 #4243  ; 刷卡密码3
AND P_EQ
CMP(20) DM13 #4144  ; 刷卡密码4
AND P_EQ
CMP(20) DM14 #4137  ; 刷卡密码5
AND P_EQ
OUT 44.07  ; 7号卡2
DIFU(13) 216.07  ; 7号卡2

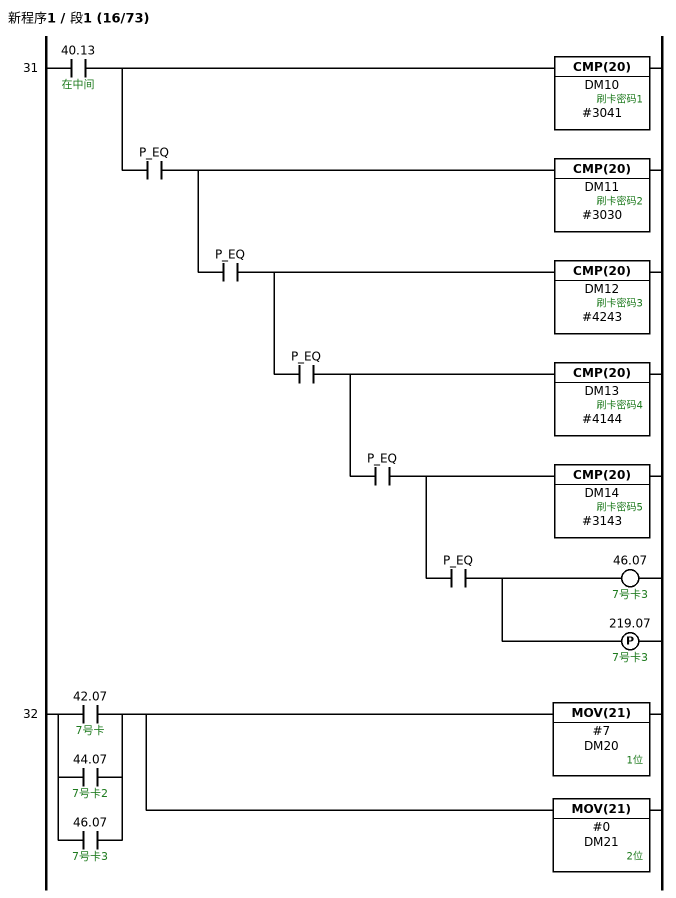
; rung 31
LD 40.13  ; 在中间
CMP(20) DM10 #3041  ; 刷卡密码1
AND P_EQ
CMP(20) DM11 #3030  ; 刷卡密码2
AND P_EQ
CMP(20) DM12 #4243  ; 刷卡密码3
AND P_EQ
CMP(20) DM13 #4144  ; 刷卡密码4
AND P_EQ
CMP(20) DM14 #3143  ; 刷卡密码5
AND P_EQ
OUT 46.07  ; 7号卡3
DIFU(13) 219.07  ; 7号卡3
; rung 32
LD 42.07  ; 7号卡
OR 44.07  ; 7号卡2
OR 46.07  ; 7号卡3
MOV(21) #7 DM20  ; 1位
MOV(21) #0 DM21  ; 2位

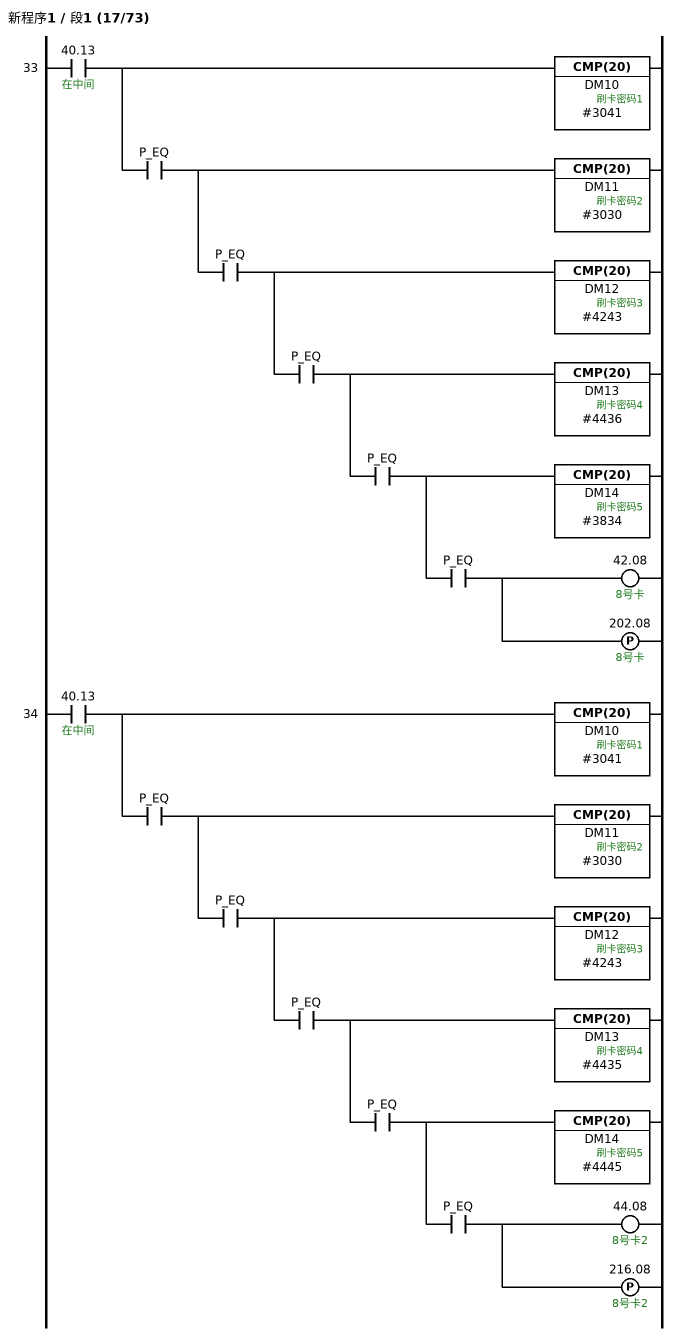
; rung 33
LD 40.13  ; 在中间
CMP(20) DM10 #3041  ; 刷卡密码1
AND P_EQ
CMP(20) DM11 #3030  ; 刷卡密码2
AND P_EQ
CMP(20) DM12 #4243  ; 刷卡密码3
AND P_EQ
CMP(20) DM13 #4436  ; 刷卡密码4
AND P_EQ
CMP(20) DM14 #3834  ; 刷卡密码5
AND P_EQ
OUT 42.08  ; 8号卡
DIFU(13) 202.08  ; 8号卡
; rung 34
LD 40.13  ; 在中间
CMP(20) DM10 #3041  ; 刷卡密码1
AND P_EQ
CMP(20) DM11 #3030  ; 刷卡密码2
AND P_EQ
CMP(20) DM12 #4243  ; 刷卡密码3
AND P_EQ
CMP(20) DM13 #4435  ; 刷卡密码4
AND P_EQ
CMP(20) DM14 #4445  ; 刷卡密码5
AND P_EQ
OUT 44.08  ; 8号卡2
DIFU(13) 216.08  ; 8号卡2

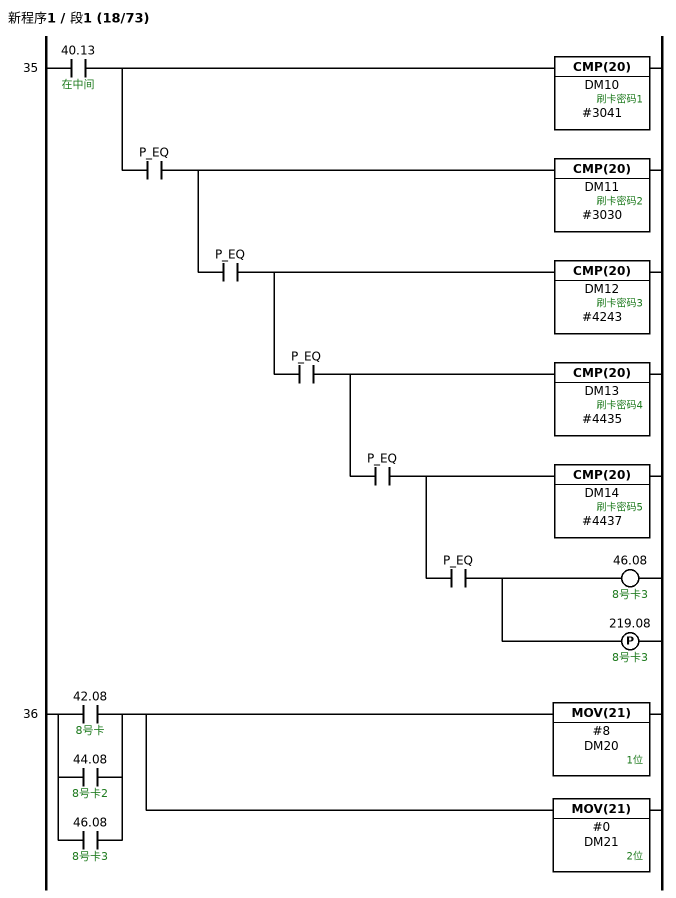
; rung 35
LD 40.13  ; 在中间
CMP(20) DM10 #3041  ; 刷卡密码1
AND P_EQ
CMP(20) DM11 #3030  ; 刷卡密码2
AND P_EQ
CMP(20) DM12 #4243  ; 刷卡密码3
AND P_EQ
CMP(20) DM13 #4435  ; 刷卡密码4
AND P_EQ
CMP(20) DM14 #4437  ; 刷卡密码5
AND P_EQ
OUT 46.08  ; 8号卡3
DIFU(13) 219.08  ; 8号卡3
; rung 36
LD 42.08  ; 8号卡
OR 44.08  ; 8号卡2
OR 46.08  ; 8号卡3
MOV(21) #8 DM20  ; 1位
MOV(21) #0 DM21  ; 2位

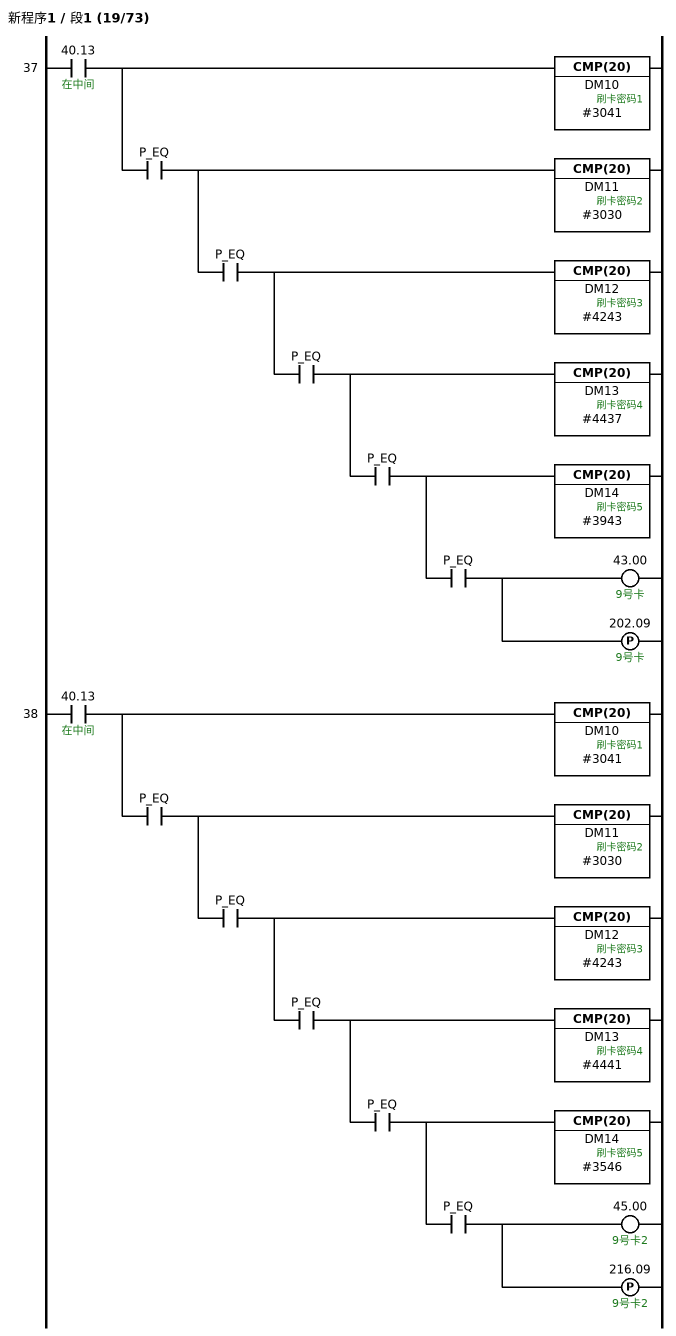
; rung 37
LD 40.13  ; 在中间
CMP(20) DM10 #3041  ; 刷卡密码1
AND P_EQ
CMP(20) DM11 #3030  ; 刷卡密码2
AND P_EQ
CMP(20) DM12 #4243  ; 刷卡密码3
AND P_EQ
CMP(20) DM13 #4437  ; 刷卡密码4
AND P_EQ
CMP(20) DM14 #3943  ; 刷卡密码5
AND P_EQ
OUT 43.00  ; 9号卡
DIFU(13) 202.09  ; 9号卡
; rung 38
LD 40.13  ; 在中间
CMP(20) DM10 #3041  ; 刷卡密码1
AND P_EQ
CMP(20) DM11 #3030  ; 刷卡密码2
AND P_EQ
CMP(20) DM12 #4243  ; 刷卡密码3
AND P_EQ
CMP(20) DM13 #4441  ; 刷卡密码4
AND P_EQ
CMP(20) DM14 #3546  ; 刷卡密码5
AND P_EQ
OUT 45.00  ; 9号卡2
DIFU(13) 216.09  ; 9号卡2

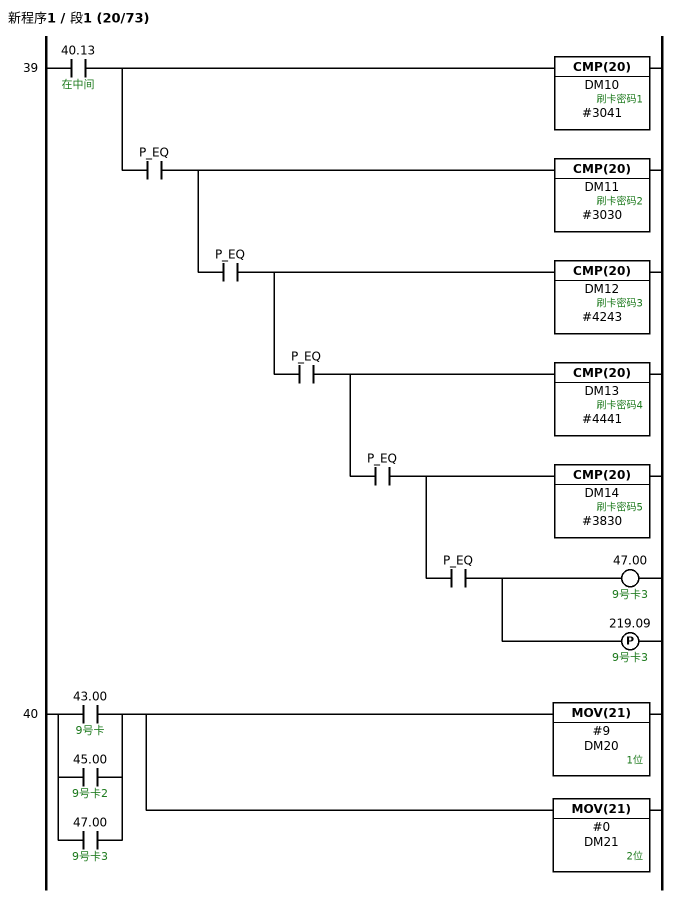
; rung 39
LD 40.13  ; 在中间
CMP(20) DM10 #3041  ; 刷卡密码1
AND P_EQ
CMP(20) DM11 #3030  ; 刷卡密码2
AND P_EQ
CMP(20) DM12 #4243  ; 刷卡密码3
AND P_EQ
CMP(20) DM13 #4441  ; 刷卡密码4
AND P_EQ
CMP(20) DM14 #3830  ; 刷卡密码5
AND P_EQ
OUT 47.00  ; 9号卡3
DIFU(13) 219.09  ; 9号卡3
; rung 40
LD 43.00  ; 9号卡
OR 45.00  ; 9号卡2
OR 47.00  ; 9号卡3
MOV(21) #9 DM20  ; 1位
MOV(21) #0 DM21  ; 2位

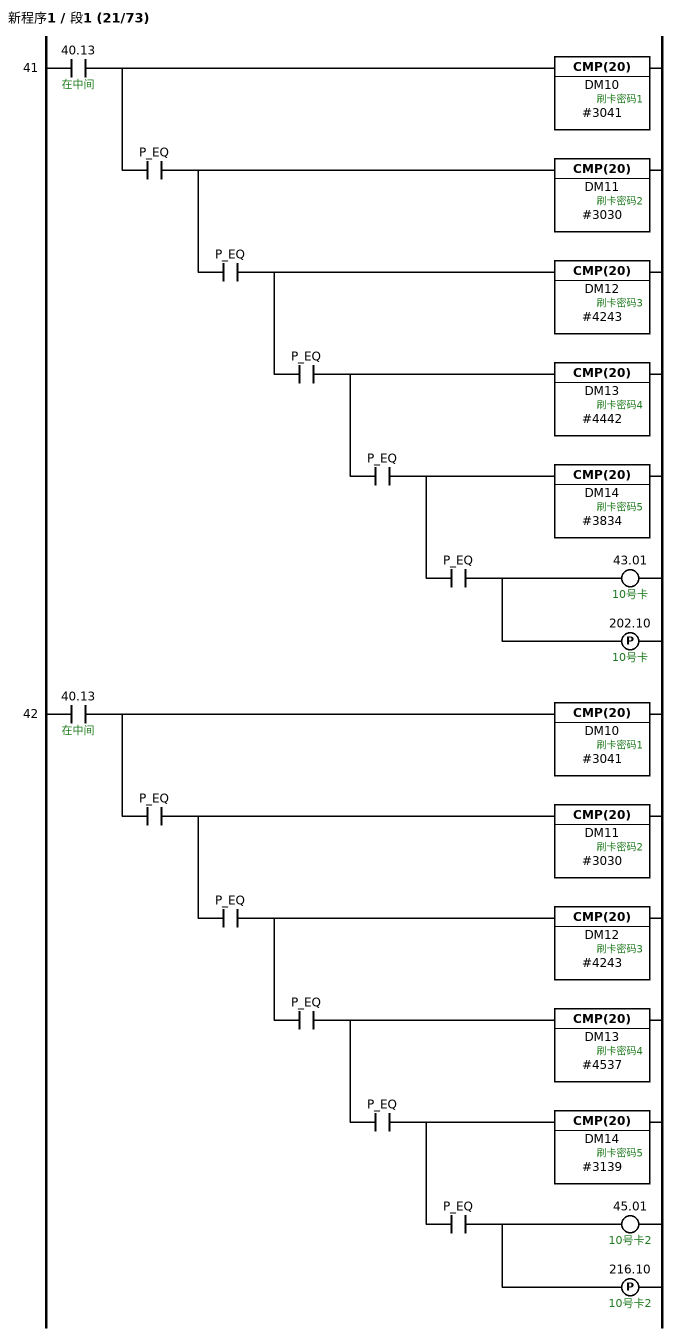
; rung 41
LD 40.13  ; 在中间
CMP(20) DM10 #3041  ; 刷卡密码1
AND P_EQ
CMP(20) DM11 #3030  ; 刷卡密码2
AND P_EQ
CMP(20) DM12 #4243  ; 刷卡密码3
AND P_EQ
CMP(20) DM13 #4442  ; 刷卡密码4
AND P_EQ
CMP(20) DM14 #3834  ; 刷卡密码5
AND P_EQ
OUT 43.01  ; 10号卡
DIFU(13) 202.10  ; 10号卡
; rung 42
LD 40.13  ; 在中间
CMP(20) DM10 #3041  ; 刷卡密码1
AND P_EQ
CMP(20) DM11 #3030  ; 刷卡密码2
AND P_EQ
CMP(20) DM12 #4243  ; 刷卡密码3
AND P_EQ
CMP(20) DM13 #4537  ; 刷卡密码4
AND P_EQ
CMP(20) DM14 #3139  ; 刷卡密码5
AND P_EQ
OUT 45.01  ; 10号卡2
DIFU(13) 216.10  ; 10号卡2

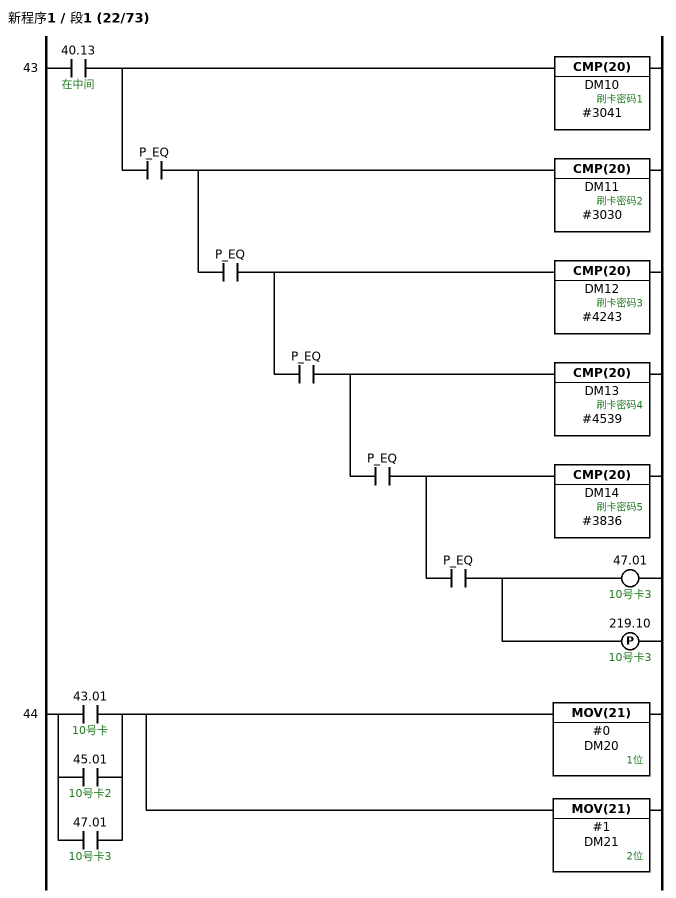
; rung 43
LD 40.13  ; 在中间
CMP(20) DM10 #3041  ; 刷卡密码1
AND P_EQ
CMP(20) DM11 #3030  ; 刷卡密码2
AND P_EQ
CMP(20) DM12 #4243  ; 刷卡密码3
AND P_EQ
CMP(20) DM13 #4539  ; 刷卡密码4
AND P_EQ
CMP(20) DM14 #3836  ; 刷卡密码5
AND P_EQ
OUT 47.01  ; 10号卡3
DIFU(13) 219.10  ; 10号卡3
; rung 44
LD 43.01  ; 10号卡
OR 45.01  ; 10号卡2
OR 47.01  ; 10号卡3
MOV(21) #0 DM20  ; 1位
MOV(21) #1 DM21  ; 2位

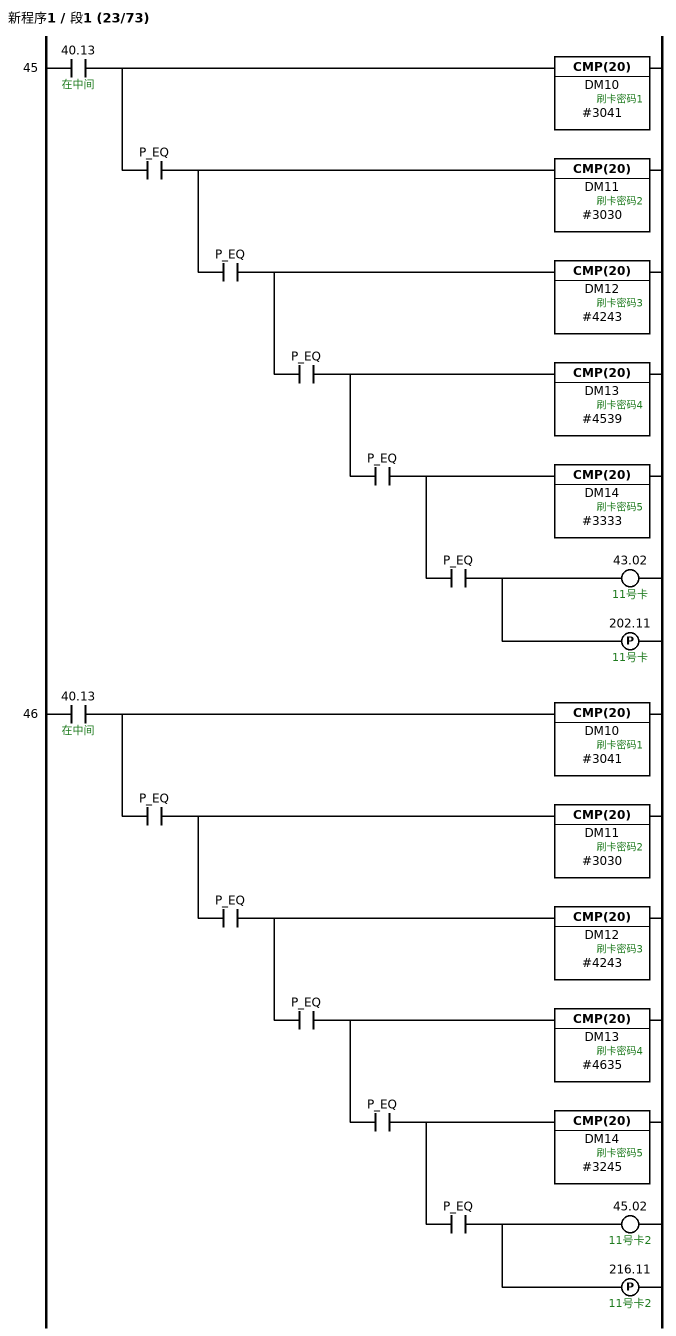
; rung 45
LD 40.13  ; 在中间
CMP(20) DM10 #3041  ; 刷卡密码1
AND P_EQ
CMP(20) DM11 #3030  ; 刷卡密码2
AND P_EQ
CMP(20) DM12 #4243  ; 刷卡密码3
AND P_EQ
CMP(20) DM13 #4539  ; 刷卡密码4
AND P_EQ
CMP(20) DM14 #3333  ; 刷卡密码5
AND P_EQ
OUT 43.02  ; 11号卡
DIFU(13) 202.11  ; 11号卡
; rung 46
LD 40.13  ; 在中间
CMP(20) DM10 #3041  ; 刷卡密码1
AND P_EQ
CMP(20) DM11 #3030  ; 刷卡密码2
AND P_EQ
CMP(20) DM12 #4243  ; 刷卡密码3
AND P_EQ
CMP(20) DM13 #4635  ; 刷卡密码4
AND P_EQ
CMP(20) DM14 #3245  ; 刷卡密码5
AND P_EQ
OUT 45.02  ; 11号卡2
DIFU(13) 216.11  ; 11号卡2

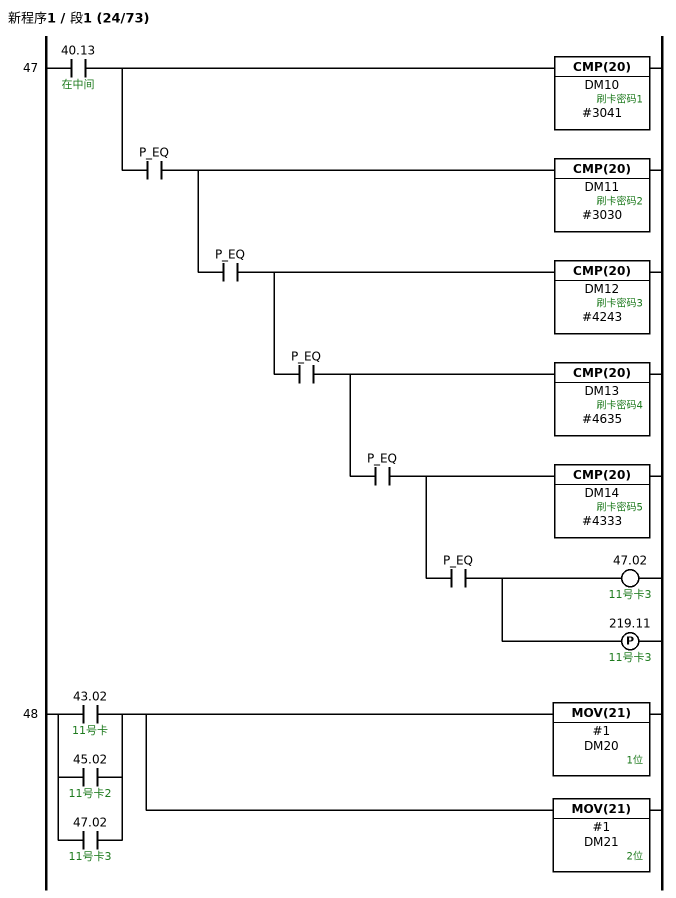
; rung 47
LD 40.13  ; 在中间
CMP(20) DM10 #3041  ; 刷卡密码1
AND P_EQ
CMP(20) DM11 #3030  ; 刷卡密码2
AND P_EQ
CMP(20) DM12 #4243  ; 刷卡密码3
AND P_EQ
CMP(20) DM13 #4635  ; 刷卡密码4
AND P_EQ
CMP(20) DM14 #4333  ; 刷卡密码5
AND P_EQ
OUT 47.02  ; 11号卡3
DIFU(13) 219.11  ; 11号卡3
; rung 48
LD 43.02  ; 11号卡
OR 45.02  ; 11号卡2
OR 47.02  ; 11号卡3
MOV(21) #1 DM20  ; 1位
MOV(21) #1 DM21  ; 2位

